// TIA Portal project "BoxWrapper" (V15)

(* hardware
DEVICE "S7-1200 station_1"  S7-1200 Station
   slot 0: "Rack_0"  S7-1200 Rack  Rack  V1.0
   slot 1: "PLC_1"  CPU 1212C DC/DC/DC  6ES7 212-1AE40-0XB0  V4.2
DEVICE "PC-System_1"  SIMATIC PC station
   slot 0: "SIMATIC PC station"  Rail  SIMATIC PC-Station  V1.0
      slot 125: "Stationmanager"  Station_Manager  V6.0.4
   slot 1: "HMI_RT_1"  WinCC RT Professional  6AV2 105-0xxxx-xxxx  15.0.0.0
   slot 2: "IE general_1"  IE General  IE_CP  V8.2.0
*)

// ===== PLC "PLC_1"  CPU 1212C DC/DC/DC =====

VAR_GLOBAL   // PLC tag table "Default tag table"
   "Start_Pb" AT %M0.1 : Bool;
   "Start_Trigger" AT %M0.0 : Bool;
   "Rotation_MotorCoil" AT %M0.2 : Bool;
   "Stop_pb" AT %M0.3 : Bool;
   "Stop_Trigger" AT %M0.4 : Bool;
   "Rotation_PX1" AT %M0.5 : Bool;
   "Rotation_Trigger1" AT %M0.6 : Bool;
   "LLSW" AT %M0.7 : Bool;
   "UpSlider_Coil" AT %M1.0 : Bool;
   "HLSW" AT %M1.1 : Bool;
   "DownSlider_Coil" AT %M1.2 : Bool;
   "Down_Trigger" AT %M1.3 : Bool;
   "Up_Trigger" AT %M1.4 : Bool;
   "Rotation_PX2" AT %M1.5 : Bool;
   "Rotation_Trigger2" AT %M1.6 : Bool;
   "Off_Trigger" AT %M1.7 : Bool;
   "EMGC" AT %M2.0 : Bool;
   "Counter_Reset" AT %M2.1 : Bool;
   "Counter_Trigger" AT %M2.2 : Bool;
   "sliderPosition" AT %MW4 : Int;
   "sliderAnimation" AT %MW6 : Int;
   "RotationAngle" AT %MW8 : Int;
   "Box90" AT %M2.3 : Bool;
   "Box180" AT %M2.4 : Bool;
   "Box270" AT %M2.5 : Bool;
   "Box45deg" AT %M2.6 : Bool;
   "Stretch_PX" AT %M2.7 : Bool;
   "Stretch_Trigger" AT %M3.0 : Bool;
   "Rerun" AT %M3.1 : Bool;
   "Rerun_Trigger" AT %M3.2 : Bool;
   "Slider_Direction" AT %MW10 : Int;
END_VAR

DATA_BLOCK "Animation1_DB"   // DB6
{ S7_Optimized_Access := 'TRUE' }
VERSION : 0.1
// stored: InstanceOfName Animation1
"Animation1"
BEGIN
END_DATA_BLOCK

// folder: System blocks/Program resources

DATA_BLOCK "Down_Counter"   // DB1
{ S7_Optimized_Access := 'TRUE' }
AUTHOR : Simatic
FAMILY : IEC
NAME : CNTR
VERSION : 1.0
// stored: InstanceOfName IEC_COUNTER
"IEC_COUNTER"
BEGIN
END_DATA_BLOCK

DATA_BLOCK "Up_Counter"   // DB2
{ S7_Optimized_Access := 'TRUE' }
AUTHOR : Simatic
FAMILY : IEC
NAME : CNTR
VERSION : 1.0
// stored: InstanceOfName IEC_COUNTER
"IEC_COUNTER"
BEGIN
END_DATA_BLOCK

DATA_BLOCK "UpTimer"   // DB3
{ S7_Optimized_Access := 'TRUE' }
AUTHOR : Simatic
FAMILY : IEC
NAME : IEC_TMR
VERSION : 1.0
// stored: InstanceOfName IEC_TIMER
"IEC_TIMER"
BEGIN
END_DATA_BLOCK

DATA_BLOCK "DownTimer"   // DB4
{ S7_Optimized_Access := 'TRUE' }
AUTHOR : Simatic
FAMILY : IEC
NAME : IEC_TMR
VERSION : 1.0
// stored: InstanceOfName IEC_TIMER
"IEC_TIMER"
BEGIN
END_DATA_BLOCK

DATA_BLOCK "RotationTimer"   // DB5
{ S7_Optimized_Access := 'TRUE' }
AUTHOR : Simatic
FAMILY : IEC
NAME : IEC_TMR
VERSION : 1.0
// stored: InstanceOfName IEC_TIMER
"IEC_TIMER"
BEGIN
END_DATA_BLOCK

DATA_BLOCK "SliderCounter"   // DB7
{ S7_Optimized_Access := 'TRUE' }
AUTHOR : Simatic
FAMILY : IEC
NAME : CNTR
VERSION : 1.0
// stored: InstanceOfName IEC_COUNTER
"IEC_COUNTER"
BEGIN
END_DATA_BLOCK

DATA_BLOCK "RotationCounter"   // DB8
{ S7_Optimized_Access := 'TRUE' }
AUTHOR : Simatic
FAMILY : IEC
NAME : CNTR
VERSION : 1.0
// stored: InstanceOfName IEC_COUNTER
"IEC_COUNTER"
BEGIN
END_DATA_BLOCK

// folder: (top level)

FUNCTION_BLOCK "Animation1"   // FB1, LAD
{ S7_Optimized_Access := 'TRUE' }
VERSION : 0.1
BEGIN

REGION Network 1
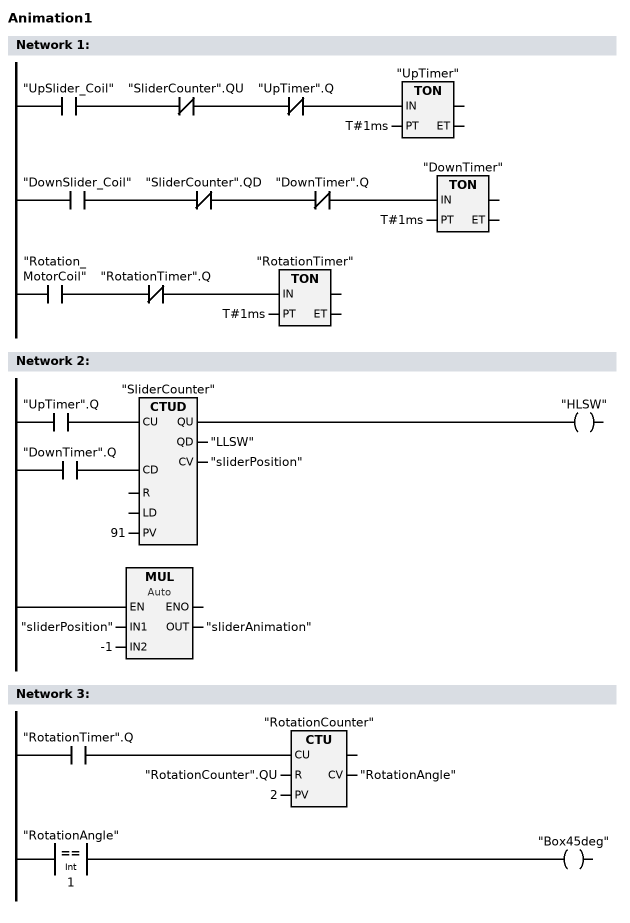
   "UpTimer".TON(IN := "UpSlider_Coil" AND NOT "SliderCounter".QU AND NOT "UpTimer".Q, PT := T#1ms);
   "DownTimer".TON(IN := "DownSlider_Coil" AND NOT "SliderCounter".QD AND NOT "DownTimer".Q, PT := T#1ms);
   "RotationTimer".TON(IN := "Rotation_MotorCoil" AND NOT "RotationTimer".Q, PT := T#1ms);
END_REGION

REGION Network 2
   "SliderCounter".CTUD(CU := "UpTimer".Q, CD := "DownTimer".Q, PV := 91, QD => "LLSW", CV => "sliderPosition");
   "HLSW" := "SliderCounter".QU;
   "sliderAnimation" := "sliderPosition" * (-1);
END_REGION

REGION Network 3
   "RotationCounter".CTU(CU := "RotationTimer".Q, R := "RotationCounter".QU, PV := 2, CV => "RotationAngle");
   "Box45deg" := "RotationAngle" = 1;
END_REGION
END_FUNCTION_BLOCK

ORGANIZATION_BLOCK "Main"   // OB1, LAD, ProgramCycle
TITLE = "Main Program Sweep (Cycle)"
{ S7_Optimized_Access := 'TRUE' }
VERSION : 0.1
   VAR_INPUT
      Initial_Call : Bool;   // Initial call of this OB
      Remanence : Bool;   // =True, if remanent data are available
   END_VAR
   VAR_TEMP   // added for the SCL form of the ladder/FBD networks
      _w1 : Bool;
      _w2 : Bool;
      _w3 : Bool;
      _w4 : Bool;
      _w5 : Bool;
      _w6 : Bool;
      _w7 : Bool;
   END_VAR
BEGIN

REGION Network 1
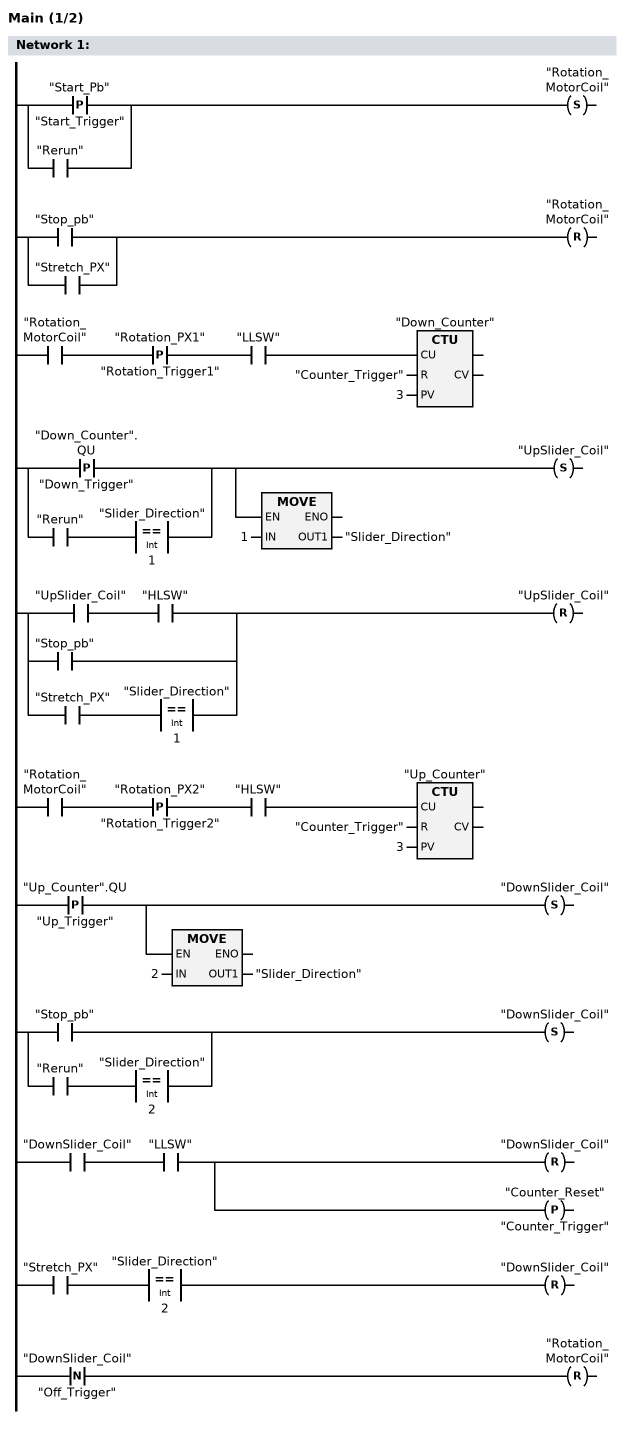
   #_w1 := "Start_Pb" AND NOT "Start_Trigger";   // rising edge of "Start_Pb"
   "Start_Trigger" := "Start_Pb";
   IF #_w1 OR "Rerun" THEN "Rotation_MotorCoil" := TRUE; END_IF;
   IF "Stop_pb" OR "Stretch_PX" THEN "Rotation_MotorCoil" := FALSE; END_IF;
   #_w2 := "Rotation_MotorCoil" AND "Rotation_PX1" AND NOT "Rotation_Trigger1";   // rising edge of "Rotation_PX1"
   "Rotation_Trigger1" := "Rotation_PX1";
   "Down_Counter".CTU(CU := #_w2 AND "LLSW", R := "Counter_Trigger", PV := 3);
   #_w3 := "Down_Counter".QU AND NOT "Down_Trigger";   // rising edge of "Down_Counter".QU
   "Down_Trigger" := "Down_Counter".QU;
   IF #_w3 OR ("Rerun" AND ("Slider_Direction" = 1)) THEN
       "UpSlider_Coil" := TRUE;
       "Slider_Direction" := 1;
   END_IF;
   IF ("UpSlider_Coil" AND "HLSW") OR "Stop_pb" OR ("Stretch_PX" AND ("Slider_Direction" = 1)) THEN
       "UpSlider_Coil" := FALSE;
   END_IF;
   #_w4 := "Rotation_MotorCoil" AND "Rotation_PX2" AND NOT "Rotation_Trigger2";   // rising edge of "Rotation_PX2"
   "Rotation_Trigger2" := "Rotation_PX2";
   "Up_Counter".CTU(CU := #_w4 AND "HLSW", R := "Counter_Trigger", PV := 3);
   #_w5 := "Up_Counter".QU AND NOT "Up_Trigger";   // rising edge of "Up_Counter".QU
   "Up_Trigger" := "Up_Counter".QU;
   IF #_w5 THEN
       "DownSlider_Coil" := TRUE;
       "Slider_Direction" := 2;
   END_IF;
   IF "Stop_pb" OR ("Rerun" AND ("Slider_Direction" = 2)) THEN "DownSlider_Coil" := TRUE; END_IF;
   #_w6 := "DownSlider_Coil" AND "LLSW";
   IF #_w6 THEN "DownSlider_Coil" := FALSE; END_IF;
   "Counter_Reset" := #_w6 AND NOT "Counter_Trigger";   // rising edge
   "Counter_Trigger" := #_w6;
   IF "Stretch_PX" AND ("Slider_Direction" = 2) THEN "DownSlider_Coil" := FALSE; END_IF;
   #_w7 := NOT "DownSlider_Coil" AND "Off_Trigger";   // falling edge of "DownSlider_Coil"
   "Off_Trigger" := "DownSlider_Coil";
   IF #_w7 THEN "Rotation_MotorCoil" := FALSE; END_IF;
END_REGION

REGION Network 2
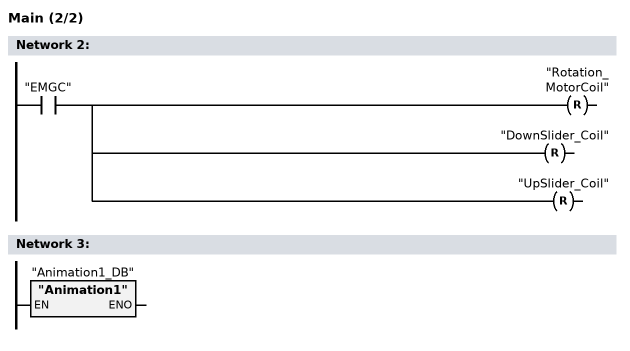
   RUNG wire#powerrail
      Contact( "EMGC" )
      wire#w1
      R_Coil( "Rotation_MotorCoil" )
   END_RUNG
   RUNG wire#w1
      R_Coil( "DownSlider_Coil" )
   END_RUNG
   RUNG wire#w1
      R_Coil( "UpSlider_Coil" )
   END_RUNG
   // the same network as SCL:
   IF "EMGC" THEN
       "Rotation_MotorCoil" := FALSE;
       "DownSlider_Coil" := FALSE;
       "UpSlider_Coil" := FALSE;
   END_IF;
END_REGION

REGION Network 3
   RUNG wire#powerrail
      "Animation1_DB"()
   END_RUNG
   // the same network as SCL:
   "Animation1_DB"();   // "Animation1"
END_REGION
END_ORGANIZATION_BLOCK

(* ===== HMI "HMI_RT_1" =====
system functions are stored by id; their names below are inferred from use
connection "PLCS7": S71200_TCP_IP, SCADA_S7_1200

HMI tags "Default tag table"
   "Start" : Bool = PLC Start_Pb AT %M0.1, 500 ms
   "Stop" : Bool = PLC Stop_pb AT %M0.3, 500 ms
   "sliderAnimation" : Int = PLC sliderAnimation AT %MW6, 500 ms
   "RotationAngle" : Int = PLC RotationAngle AT %MW8, 500 ms
   "RotationPX1" : Bool = PLC Rotation_PX1 AT %M0.5, 500 ms
   "RotationPX2" : Bool = PLC Rotation_PX2 AT %M1.5, 500 ms
   "AnotherBox" : Bool = PLC Box45deg AT %M2.6, 500 ms
   "StretchPX" : Bool = PLC Stretch_PX AT %M2.7, 500 ms
   "Rerun" : Bool = PLC Rerun AT %M3.1, 500 ms
   "EMGC" : Bool = PLC EMGC AT %M2.0, 500 ms

screen "Screen_1" 500x500
   on PressLeft: SetBit("RotationPX2")
   on ReleaseLeft: ResetBit("RotationPX2")
   Button "Button_1" at 9,465 size 80x26; TextOff 'START'
      on PressLeft: SetBit("Start")
      on ReleaseLeft: ResetBit("Start")
   TextField "Text field_1" at 174,9 size 124x23; Text 'Box Wrapper'
   Button "Button_2" at 94,465 size 80x26; TextOff 'STOP'
      on PressLeft: SetBit("Stop")
      on ReleaseLeft: ResetBit("Stop")
   Button "Button_3" at 414,465 size 80x27; TextOff 'EXIT'
      on Click: StopRuntime(0)
   Group "Group" at 42,351 size 175x32
      DirectMovement <- "sliderAnimation"
   Group "Group_1" at 27,249 size 43x11
   Group "Group_2" at 27,377 size 43x11
   Rectangle "Rectangle_10" at 289,249 size 140x128
      Visibility <- "AnotherBox"
   TextField "Text field_2" at 53,212 size 114x16; Text 'Upper Limit Sensor'
   TextField "Text field_3" at 25,406 size 114x16; Text 'Lower Limit Sensor'
   RoundButton "Round button_1" at 420,98 size 48x48; Text 'PX1'
      on PressLeft: SetBit("RotationPX1")
      on ReleaseLeft: ResetBit("RotationPX1")
   RoundButton "Round button_2" at 420,153 size 48x48; Text 'PX2'
      on PressLeft: SetBit("RotationPX2")
      on ReleaseLeft: ResetBit("RotationPX2")
   Polygon "Polygon_1" at 271,223 size 182x181
      Visibility <- "AnotherBox"
   TextField "Text field_4" at 305,115 size 129x16; Text 'Lower Proximity SW'
   TextField "Text field_5" at 306,169 size 114x16; Text 'Upper Proximity SW'
   Group "Group_3" at 422,294 size 43x32
   TextField "Text field_7" at 127,117 size 129x16; Text 'Stretch Proximity SW'
   RoundButton "Round button_3" at 70,98 size 48x48; Text 'SX'
      on PressLeft: SetBit("StretchPX")
      on ReleaseLeft: ResetBit("StretchPX")
   RoundButton "Round button_4" at 70,153 size 48x48; Text 'RERUN'
      on PressLeft: SetBit("Rerun")
      on ReleaseLeft: ResetBit("Rerun")
   RoundButton "Round button_5" at 265,459 size 38x38; Text 'EMGC'
      on PressLeft: SetBit("EMGC")
      on ReleaseLeft: ResetBit("EMGC")
*)